PROGRAM MAIN
VAR
	fbStateMachine				:	FB_StateMachine();
	fbHeatPumpIO				:	FB_HeatpumpIO();
	sState						:	STRING;
	bOnButtonPressed    		: 	BOOL;
	bOffButtonPressed			: 	BOOL;
	bConfirmationButtonPressed	: 	BOOL;
END_VAR

fbStateMachine(	bOnButtonPressed				:= bOnButtonPressed,
				bOffButtonPressed				:= bOffButtonPressed,
				bConfirmationButtonPressed		:= bConfirmationButtonPressed);
				
fbHeatPumpIO();				
	
sState : fbStateMachine.ipState.Description;
bOnButtonPressed			:= FALSE;
bOffButtonPressed			:= FALSE;
bConfirmationButtonPressed	:= FALSE;

END_PROGRAM

(* stored: Version 1.1.0.1
   POU MAIN: Id {e3e9ea5b-aaa6-4abd-9e50-1f99907708dc}, SpecialFunc None *)
